// TIA Portal V16 export
// export: Created 2026-06-17T18:28:32.8881869Z, ExportSetting WithDefaults, DisplayName Totally Integrated Automation Portal, DisplayVersion V16 Update 8, DisplayName TIA Portal Version Control Interface, DisplayVersion V16 Update 8, DisplayName TIA Portal Openness, DisplayVersion V16 Update 8, DisplayName SINAMICS Startdrive Advanced, DisplayVersion V16, DisplayName SINAMICS Startdrive G130, G150, S120, S150, SINAMICS MV, S210, DisplayVersion V16, DisplayName SINAMICS Startdrive G110M, G120, G120C, G120D, G120P, DisplayVersion V16, DisplayName STEP 7 Professional, DisplayVersion V16 Update 8, DisplayName STEP 7 Safety, DisplayVersion V16 Update 7, DisplayName WinCC Advanced, DisplayVersion V16 Update 8
Screen "Motor_Control"  1280x800, Number=1
  ScreenLayer 
    IOField "IO_Speed" at 280,320 size 160x44  DataFormat=Decimal, FormatPattern=9999999, Mode=InOutput
    Button "BTN_Reset" at 440,140 size 130x56  Mode=Text, HelpText="复位", TextOff="Text", TextOn="Text"
    SymbolicIOField "SIO_Mode" at 280,400 size 160x44  CountVisibleItems=3, Mode=InOutput, OnValue=1, TextOff="0", TextOn="1"
    Circle "LMP_Fault" at 880,148 size 48x48
    TextField "TXT_Title" at 440,30 size 400x48  Text="电机控制画面Text"
